# EPICS autosave request: ADPixirad/iocs/pixiradIOC/iocBoot/iocPixirad/auto_settings.req
file "pixirad_settings.req",      P=$(P),  R=cam1:
file "NDStdArrays_settings.req",  P=$(P),  R=image1:
file "commonPlugin_settings.req", P=$(P)
